(* CoDeSys 2.3.9.45 project: FUP.pro *)
(* Libraries: Standard.lib 2.12.10 14:48:34, SYSLIBCALLBACK.LIB 2.12.10 14:48:32 *)

(* PLC configuration (modules and I/O channels)
K-Bus [K_Bus] node 0, in %IB0 out %QB0
Fieldbus variables [FB_VARS] node 1, in %IB0 out %QB0
Flag variables [FLAG_VARS] node 2, in %IB0 out %QB0
Modbus-Master [MB_MASTER] node 3, in %IB0 out %QB0
*)

(* POU PLC_PRG, FBD *)
PROGRAM PLC_PRG

VAR
	K1: BOOL;
	K2: BOOL;
END_VAR

VAR_INPUT
	S8: BOOL;
	S12: BOOL;
	S11: BOOL;
	S22: BOOL;
	S21: BOOL;
END_VAR
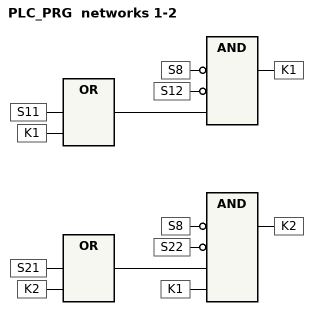
_FBD_ (* Function Block Diagram *)
NETWORK 1
	AND(NOT S8, NOT S12, OR(S11, K1)) => K1
NETWORK 2
	AND(NOT S8, NOT S22, OR(S21, K2), K1) => K2
_END_FBD_
(* the same logic as Structured Text *)
(* Network 1 *)
K1 := NOT S8 AND NOT S12 AND (S11 OR K1);
(* Network 2 *)
K2 := NOT S8 AND NOT S22 AND (S21 OR K2) AND K1;
END_PROGRAM
